Staubli VAL3: connectTo.pgx

public program connectTo(string x_sIp, num x_nRack, num x_nSlot)
  local string l_sTempBin
  local string l_sRes
  local num l_nTempDec
begin

  //set connection parameters
  sioCtrl(sTCPclient, "target", x_sIp)

  nLocalTSAP_HI = 1
  nLocalTSAP_LO = 0

  //nRemoteTSAP_HI
  l_sTempBin=""
  call bitOp:DecToBin(((nConnType*256) + (x_nRack*32) + x_nSlot), l_sTempBin)
  call bitOp:shiftRight(l_sTempBin, 8)
  l_nTempDec=0
  call bitOp:BinToDec(l_sTempBin, l_nTempDec)
  nRemoteTSAP_HI=l_nTempDec

  //nRemoteTSAP_LO
  l_sTempBin=""
  call bitOp:DecToBin(((nConnType*256) + (x_nRack*32) + x_nSlot), l_sTempBin)
  call bitOp:boolAnd(l_sTempBin, "0000000011111111", l_sRes)
  l_nTempDec=0
  call bitOp:BinToDec(l_sRes, l_nTempDec)
  nRemoteTSAP_LO=l_nTempDec

  call setLastError(nNoErrors)
  if !bConnected
    call TCPConnect()
    if nLastError==nNoErrors
      call ISOConnect()
      if nLastError==nNoErrors
        //putln("connected to plc!")
        call negotPduLength()
      endIf
    endIf
  endIf

  if nLastError==nNoErrors
    bConnected=true
  endIf

end
